// TIA Portal V20 export
DATA_BLOCK "DB_StandardAccess"   // DB48
{ S7_Optimized_Access := 'FALSE' }
VERSION : 0.1
// stored: AutoNumber true, DBAccessibleFromOPCUA true, IsOnlyStoredInLoadMemory false, IsWriteProtectedInAS false
   VAR
      RegisterStore : Array[0..67] of Byte;
   END_VAR
BEGIN
END_DATA_BLOCK
